FUNCTION_BLOCK RT_E_SWITCH (* Split an event to two event chain branches *)
  (* Standard: 61499-2 *)
  (* Version 0.0, 2008-07-10, 4DIAC-IDE, 4DIAC-Consortium *)
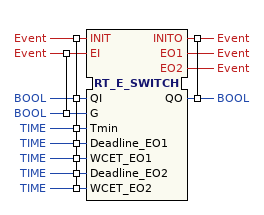
  EVENT_INPUT
    INIT WITH QI, Tmin, Deadline_EO1, WCET_EO1, Deadline_EO2, WCET_EO2;
    EI WITH G; (* Input event *)
  END_EVENT
  EVENT_OUTPUT
    INITO WITH QO;
    EO1; (* First output event *)
    EO2; (* Second output event,etc. *)
  END_EVENT
  VAR_INPUT
    QI : BOOL;
    G : BOOL;
    Tmin : TIME;
    Deadline_EO1 : TIME;
    WCET_EO1 : TIME;
    Deadline_EO2 : TIME;
    WCET_EO2 : TIME;
  END_VAR
  VAR_OUTPUT
    QO : BOOL;
  END_VAR
END_FUNCTION_BLOCK
